// TIA Portal V17 export
// export: Created 2024-09-02T12:49:54.6510911Z, ExportSetting WithDefaults, DisplayName Totally Integrated Automation Portal, DisplayVersion V17, DisplayName TIA Portal Openness, DisplayVersion V17, DisplayName TIA Portal Version Control Interface, DisplayVersion V17, DisplayName STEP 7 Professional, DisplayVersion V17, DisplayName STEP 7 Safety, DisplayVersion V17, DisplayName WinCC Professional, DisplayVersion V17
FUNCTION "AnwFC_ZP_PNIO_Diagnose" : Void   // FC1296, LAD
TITLE = PNIO Diagnostics / PNIO Diagnose
{ S7_Optimized_Access := 'TRUE' }
AUTHOR : OlegFuehrus
FAMILY : BA
NAME : BA
VERSION : 0.1
// stored: AutoNumber true, IsIECCheckEnabled false, SetENOAutomatically false, UDAEnableTagReadback false
   VAR_TEMP
      PNIO_NR : Int;
      _Ret_Val : Int;
   END_VAR
   VAR_TEMP   // added for the SCL form of the ladder/FBD networks
      _w1 : Bool;
      _w2 : Bool;
   END_VAR
BEGIN

REGION Network 1: Profinet Diagnostics Reading data / Profinet Diagnose Daten Einlesen
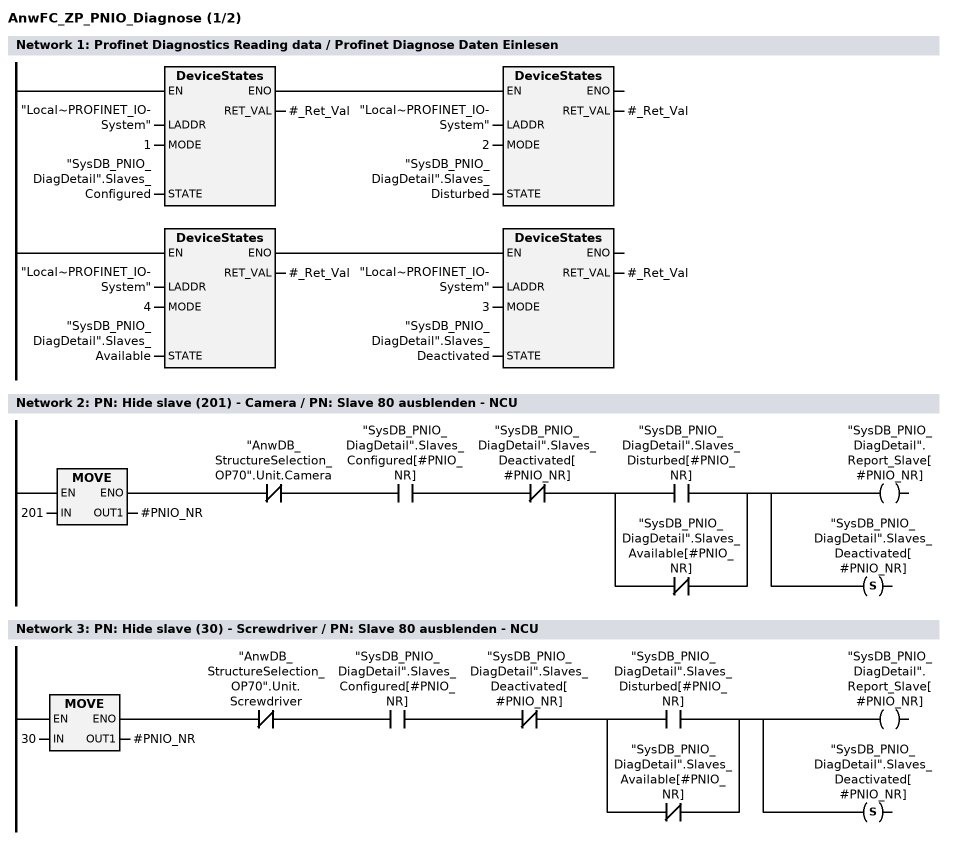
   RUNG wire#powerrail
      DeviceStates(LADDR := "Local~PROFINET_IO-System", MODE := 1, STATE := "SysDB_PNIO_DiagDetail".Slaves_Configured, Ret_Val => #_Ret_Val)
      DeviceStates(LADDR := "Local~PROFINET_IO-System", MODE := 2, STATE := "SysDB_PNIO_DiagDetail".Slaves_Disturbed, Ret_Val => #_Ret_Val)
   END_RUNG
   RUNG wire#powerrail
      DeviceStates(LADDR := "Local~PROFINET_IO-System", MODE := 4, STATE := "SysDB_PNIO_DiagDetail".Slaves_Available, Ret_Val => #_Ret_Val)
      DeviceStates(LADDR := "Local~PROFINET_IO-System", MODE := 3, STATE := "SysDB_PNIO_DiagDetail".Slaves_Deactivated, Ret_Val => #_Ret_Val)
   END_RUNG
   // the same network as SCL:
   #_Ret_Val := DeviceStates(LADDR := "Local~PROFINET_IO-System",
                           MODE := 1,
                           STATE := "SysDB_PNIO_DiagDetail".Slaves_Configured,
                           ENO => #_w1);
   IF #_w1 THEN
       #_Ret_Val := DeviceStates(LADDR := "Local~PROFINET_IO-System",
                               MODE := 2,
                               STATE := "SysDB_PNIO_DiagDetail".Slaves_Disturbed);
   END_IF;
   #_Ret_Val := DeviceStates(LADDR := "Local~PROFINET_IO-System",
                           MODE := 4,
                           STATE := "SysDB_PNIO_DiagDetail".Slaves_Available,
                           ENO => #_w2);
   IF #_w2 THEN
       #_Ret_Val := DeviceStates(LADDR := "Local~PROFINET_IO-System",
                               MODE := 3,
                               STATE := "SysDB_PNIO_DiagDetail".Slaves_Deactivated);
   END_IF;
END_REGION

REGION Network 2: PN: Hide slave (201) - Camera / PN: Slave 80 ausblenden - NCU
   RUNG wire#powerrail
      Move(in := 201, out1 => #PNIO_NR)
      I_Contact( "AnwDB_StructureSelection_OP70".Unit.Camera )
      Contact( "SysDB_PNIO_DiagDetail".Slaves_Configured[#PNIO_NR] )
      I_Contact( "SysDB_PNIO_DiagDetail".Slaves_Deactivated[#PNIO_NR] )
      wire#w1
      Contact( "SysDB_PNIO_DiagDetail".Slaves_Disturbed[#PNIO_NR] )
      wire#w2
      Coil( "SysDB_PNIO_DiagDetail".Report_Slave[#PNIO_NR] )
   END_RUNG
   RUNG wire#w1
      I_Contact( "SysDB_PNIO_DiagDetail".Slaves_Available[#PNIO_NR] )
   END_RUNG wire#w2
   RUNG wire#w2
      S_Coil( "SysDB_PNIO_DiagDetail".Slaves_Deactivated[#PNIO_NR] )
   END_RUNG
   // the same network as SCL:
   #PNIO_NR := 201;
   #_w1 := NOT "AnwDB_StructureSelection_OP70".Unit.Camera AND "SysDB_PNIO_DiagDetail".Slaves_Configured[#PNIO_NR] AND NOT "SysDB_PNIO_DiagDetail".Slaves_Deactivated[#PNIO_NR] AND ("SysDB_PNIO_DiagDetail".Slaves_Disturbed[#PNIO_NR] OR NOT "SysDB_PNIO_DiagDetail".Slaves_Available[#PNIO_NR]);
   "SysDB_PNIO_DiagDetail".Report_Slave[#PNIO_NR] := NOT "AnwDB_StructureSelection_OP70".Unit.Camera AND "SysDB_PNIO_DiagDetail".Slaves_Configured[#PNIO_NR] AND NOT "SysDB_PNIO_DiagDetail".Slaves_Deactivated[#PNIO_NR] AND ("SysDB_PNIO_DiagDetail".Slaves_Disturbed[#PNIO_NR] OR NOT "SysDB_PNIO_DiagDetail".Slaves_Available[#PNIO_NR]);
   IF #_w1 THEN "SysDB_PNIO_DiagDetail".Slaves_Deactivated[#PNIO_NR] := TRUE; END_IF;
END_REGION

REGION Network 3: PN: Hide slave (30) - Screwdriver / PN: Slave 80 ausblenden - NCU
   RUNG wire#powerrail
      Move(in := 30, out1 => #PNIO_NR)
      I_Contact( "AnwDB_StructureSelection_OP70".Unit.Screwdriver )
      Contact( "SysDB_PNIO_DiagDetail".Slaves_Configured[#PNIO_NR] )
      I_Contact( "SysDB_PNIO_DiagDetail".Slaves_Deactivated[#PNIO_NR] )
      wire#w1
      Contact( "SysDB_PNIO_DiagDetail".Slaves_Disturbed[#PNIO_NR] )
      wire#w2
      Coil( "SysDB_PNIO_DiagDetail".Report_Slave[#PNIO_NR] )
   END_RUNG
   RUNG wire#w1
      I_Contact( "SysDB_PNIO_DiagDetail".Slaves_Available[#PNIO_NR] )
   END_RUNG wire#w2
   RUNG wire#w2
      S_Coil( "SysDB_PNIO_DiagDetail".Slaves_Deactivated[#PNIO_NR] )
   END_RUNG
   // the same network as SCL:
   #PNIO_NR := 30;
   #_w1 := NOT "AnwDB_StructureSelection_OP70".Unit.Screwdriver AND "SysDB_PNIO_DiagDetail".Slaves_Configured[#PNIO_NR] AND NOT "SysDB_PNIO_DiagDetail".Slaves_Deactivated[#PNIO_NR] AND ("SysDB_PNIO_DiagDetail".Slaves_Disturbed[#PNIO_NR] OR NOT "SysDB_PNIO_DiagDetail".Slaves_Available[#PNIO_NR]);
   "SysDB_PNIO_DiagDetail".Report_Slave[#PNIO_NR] := NOT "AnwDB_StructureSelection_OP70".Unit.Screwdriver AND "SysDB_PNIO_DiagDetail".Slaves_Configured[#PNIO_NR] AND NOT "SysDB_PNIO_DiagDetail".Slaves_Deactivated[#PNIO_NR] AND ("SysDB_PNIO_DiagDetail".Slaves_Disturbed[#PNIO_NR] OR NOT "SysDB_PNIO_DiagDetail".Slaves_Available[#PNIO_NR]);
   IF #_w1 THEN "SysDB_PNIO_DiagDetail".Slaves_Deactivated[#PNIO_NR] := TRUE; END_IF;
END_REGION

REGION Network 4: Evaluate Profinet / Profinet Auswerten
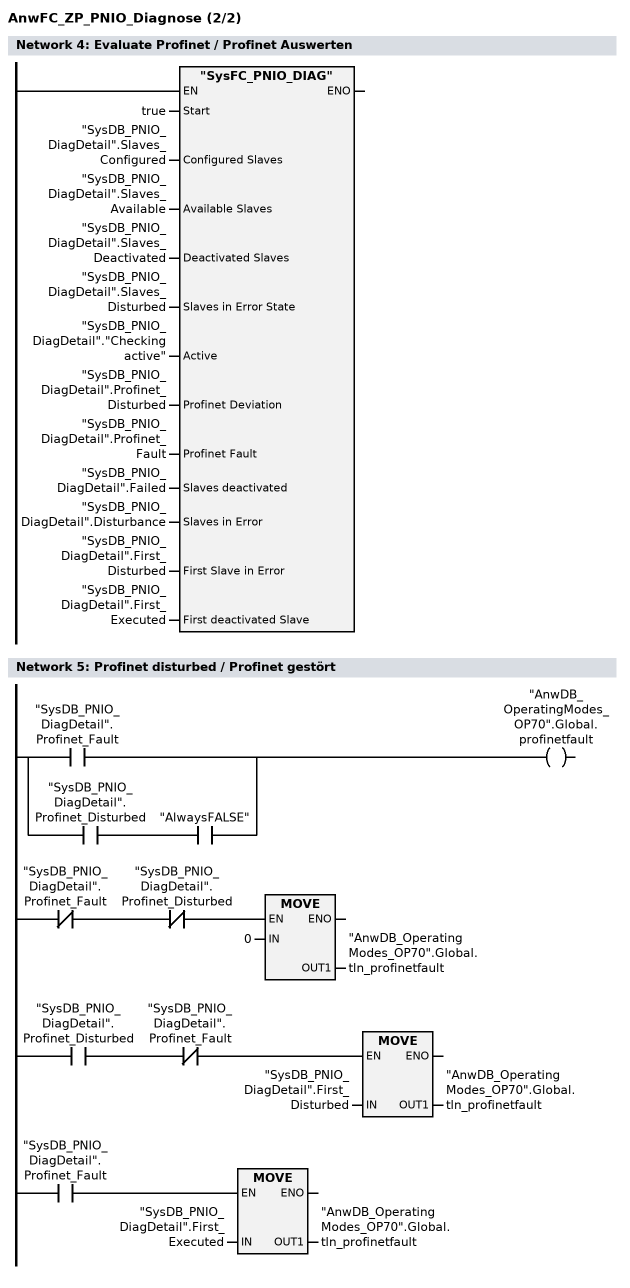
   RUNG wire#powerrail
      "SysFC_PNIO_DIAG"(Start := true, "Configured Slaves" := "SysDB_PNIO_DiagDetail".Slaves_Configured, "Available Slaves" := "SysDB_PNIO_DiagDetail".Slaves_Available, "Deactivated Slaves" := "SysDB_PNIO_DiagDetail".Slaves_Deactivated, "Slaves in Error State" := "SysDB_PNIO_DiagDetail".Slaves_Disturbed, Active := "SysDB_PNIO_DiagDetail"."Checking active", "Profinet Deviation" := "SysDB_PNIO_DiagDetail".Profinet_Disturbed, "Profinet Fault" := "SysDB_PNIO_DiagDetail".Profinet_Fault, "Slaves deactivated" := "SysDB_PNIO_DiagDetail".Failed, "Slaves in Error" := "SysDB_PNIO_DiagDetail".Disturbance, "First Slave in Error" := "SysDB_PNIO_DiagDetail".First_Disturbed, "First deactivated Slave" := "SysDB_PNIO_DiagDetail".First_Executed)
   END_RUNG
   // the same network as SCL:
   "SysFC_PNIO_DIAG"(Start := true,
                     "Configured Slaves" := "SysDB_PNIO_DiagDetail".Slaves_Configured,
                     "Available Slaves" := "SysDB_PNIO_DiagDetail".Slaves_Available,
                     "Deactivated Slaves" := "SysDB_PNIO_DiagDetail".Slaves_Deactivated,
                     "Slaves in Error State" := "SysDB_PNIO_DiagDetail".Slaves_Disturbed,
                     Active := "SysDB_PNIO_DiagDetail"."Checking active",
                     "Profinet Deviation" := "SysDB_PNIO_DiagDetail".Profinet_Disturbed,
                     "Profinet Fault" := "SysDB_PNIO_DiagDetail".Profinet_Fault,
                     "Slaves deactivated" := "SysDB_PNIO_DiagDetail".Failed,
                     "Slaves in Error" := "SysDB_PNIO_DiagDetail".Disturbance,
                     "First Slave in Error" := "SysDB_PNIO_DiagDetail".First_Disturbed,
                     "First deactivated Slave" := "SysDB_PNIO_DiagDetail".First_Executed);
END_REGION

REGION Network 5: Profinet disturbed / Profinet gestört
   RUNG wire#powerrail
      Contact( "SysDB_PNIO_DiagDetail".Profinet_Fault )
      wire#w1
      Coil( "AnwDB_OperatingModes_OP70".Global.profinetfault )
   END_RUNG
   RUNG wire#powerrail
      Contact( "SysDB_PNIO_DiagDetail".Profinet_Disturbed )
      Contact( "AlwaysFALSE" )
   END_RUNG wire#w1
   RUNG wire#powerrail
      I_Contact( "SysDB_PNIO_DiagDetail".Profinet_Fault )
      I_Contact( "SysDB_PNIO_DiagDetail".Profinet_Disturbed )
      Move(in := 0, out1 => "AnwDB_OperatingModes_OP70".Global.tln_profinetfault)
   END_RUNG
   RUNG wire#powerrail
      Contact( "SysDB_PNIO_DiagDetail".Profinet_Disturbed )
      I_Contact( "SysDB_PNIO_DiagDetail".Profinet_Fault )
      Move(in := "SysDB_PNIO_DiagDetail".First_Disturbed, out1 => "AnwDB_OperatingModes_OP70".Global.tln_profinetfault)
   END_RUNG
   RUNG wire#powerrail
      Contact( "SysDB_PNIO_DiagDetail".Profinet_Fault )
      Move(in := "SysDB_PNIO_DiagDetail".First_Executed, out1 => "AnwDB_OperatingModes_OP70".Global.tln_profinetfault)
   END_RUNG
   // the same network as SCL:
   "AnwDB_OperatingModes_OP70".Global.profinetfault := "SysDB_PNIO_DiagDetail".Profinet_Fault OR ("SysDB_PNIO_DiagDetail".Profinet_Disturbed AND "AlwaysFALSE");
   IF NOT "SysDB_PNIO_DiagDetail".Profinet_Fault AND NOT "SysDB_PNIO_DiagDetail".Profinet_Disturbed THEN
       "AnwDB_OperatingModes_OP70".Global.tln_profinetfault := 0;
   END_IF;
   IF "SysDB_PNIO_DiagDetail".Profinet_Disturbed AND NOT "SysDB_PNIO_DiagDetail".Profinet_Fault THEN
       "AnwDB_OperatingModes_OP70".Global.tln_profinetfault := "SysDB_PNIO_DiagDetail".First_Disturbed;
   END_IF;
   IF "SysDB_PNIO_DiagDetail".Profinet_Fault THEN
       "AnwDB_OperatingModes_OP70".Global.tln_profinetfault := "SysDB_PNIO_DiagDetail".First_Executed;
   END_IF;
END_REGION
END_FUNCTION
